PROGRAM AxisServoCtrl_SlowPull
VAR

	ArmSlowPullFB					: fbSlowPullAxisCtrl;
	SlowPullPosStart				: CMP_OC_W1;
	SlowPullTimer					: TON;

END_VAR

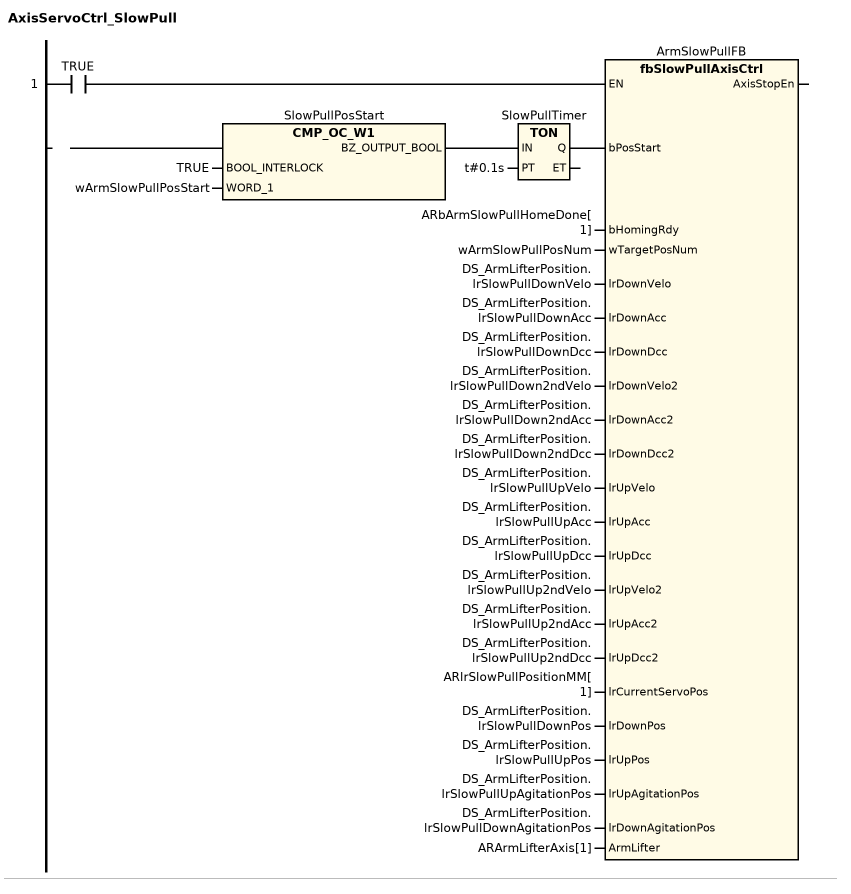
// NETWORK 1
SlowPullPosStart(BOOL_INTERLOCK := TRUE, WORD_1 := wArmSlowPullPosStart); // CMP_OC_W1
SlowPullTimer(IN := SlowPullPosStart.BZ_OUTPUT_BOOL, PT := t#0.1s); // TON
ArmSlowPullFB(
    bPosStart := SlowPullTimer.Q,
    bHomingRdy := ARbArmSlowPullHomeDone[1],
    wTargetPosNum := wArmSlowPullPosNum,
    lrDownVelo := DS_ArmLifterPosition.lrSlowPullDownVelo,
    lrDownAcc := DS_ArmLifterPosition.lrSlowPullDownAcc,
    lrDownDcc := DS_ArmLifterPosition.lrSlowPullDownDcc,
    lrDownVelo2 := DS_ArmLifterPosition.lrSlowPullDown2ndVelo,
    lrDownAcc2 := DS_ArmLifterPosition.lrSlowPullDown2ndAcc,
    lrDownDcc2 := DS_ArmLifterPosition.lrSlowPullDown2ndDcc,
    lrUpVelo := DS_ArmLifterPosition.lrSlowPullUpVelo,
    lrUpAcc := DS_ArmLifterPosition.lrSlowPullUpAcc,
    lrUpDcc := DS_ArmLifterPosition.lrSlowPullUpDcc,
    lrUpVelo2 := DS_ArmLifterPosition.lrSlowPullUp2ndVelo,
    lrUpAcc2 := DS_ArmLifterPosition.lrSlowPullUp2ndAcc,
    lrUpDcc2 := DS_ArmLifterPosition.lrSlowPullUp2ndDcc,
    lrCurrentServoPos := ARlrSlowPullPositionMM[1],
    lrDownPos := DS_ArmLifterPosition.lrSlowPullDownPos,
    lrUpPos := DS_ArmLifterPosition.lrSlowPullUpPos,
    lrUpAgitationPos := DS_ArmLifterPosition.lrSlowPullUpAgitationPos,
    lrDownAgitationPos := DS_ArmLifterPosition.lrSlowPullDownAgitationPos,
    ArmLifter := ARArmLifterAxis[1]); // fbSlowPullAxisCtrl

END_PROGRAM

(* stored: Version 1.1.0.1, ProductVersion 3.1.4024.12
   POU AxisServoCtrl_SlowPull: Id {68e4b1b0-8af1-4fb8-a398-5765d9a0428f}, SpecialFunc None *)
